Fanuc KAREL source: kd00014.KL

-- PROVISIONAL review KL for V770-1; original PC SHA256 c1a99c497574bef35d106d7975e9bf64cf9c31f88b8969fe900c460492d09e46
-- Incomplete behavior may be omitted. Consult companion uncertainty JSON. Do not deploy.
PROGRAM KD00014
%NOLOCKGROUP
VAR
  I : INTEGER
  J : INTEGER
  B : BOOLEAN
  R : REAL
  S : STRING[80]
BEGIN
  -- UNRESOLVED_PC offsets 5-9; opcodes 9C,9D,1A
  -- UNRESOLVED_PC offsets 14-18; opcodes 7F
END KD00014
